FUNCTION_BLOCK Test_AggregateResult_Ready EXTENDS T_UnitTestBase
VAR
    ResultAggregate : T_ResultAggregate;
    Execution1      : T_Execution;
    Execution2      : T_Execution;
    Execution3      : T_Execution;
END_VAR

METHOD Init
SUPER^.Init();

Execution1.FB_init(FALSE,FALSE);
Execution2.FB_init(FALSE,FALSE);
Execution3.FB_init(FALSE,FALSE);
END_METHOD

{attribute 'analysis' := '-33'} // inhibit unused variable warning
METHOD RunTest
ResultAggregate.ClearResults();

ResultAggregate.AddResult(Execution1);
ResultAggregate.AddResult(Execution2);
ResultAggregate.AddResult(Execution3);

AssertIsTrue(Condition := ResultAggregate.Ready = TRUE,
             Message   := 'ResultAggregate.Ready is not true');

Execution1.Start();
Execution1.SetBusy();

AssertIsTrue(Condition := ResultAggregate.Ready = FALSE,
             Message   := 'ResultAggregate.Ready is not false');

TestCompleted := TRUE;
END_METHOD

END_FUNCTION_BLOCK

(* stored: Version 1.1.0.1, ProductVersion 3.1.4024.12
   POU Test_AggregateResult_Ready: Id {72ffb8f8-97c0-47ff-a4ef-9542a58dc31a}, SpecialFunc None
   Method Init: Id {60cf34be-11ea-407e-96de-44b3e807ddb1}
   Method RunTest: Id {750c171c-decc-468d-90f1-12d23adfe68a} *)
